// TIA Portal V19 export
TYPE "LAF_typeChecksumCatWord"
TITLE = Structure PLC checksum cat word / Struktur PLC Checksum cat Word
// Type contains the structure for RetVal values. / PLC Checksum
// stored: Access Published
   STRUCT
      standard { ExternalAccessible := 'False'; ExternalVisible := 'False'; ExternalWritable := 'False'} : Word;   // Standard
      safety { ExternalAccessible := 'False'; ExternalVisible := 'False'; ExternalWritable := 'False'} : Word;   // Safety
      textlists { ExternalAccessible := 'False'; ExternalVisible := 'False'; ExternalWritable := 'False'} : Word;   // Textlisten / Textlists
   END_STRUCT;
END_TYPE
